{attribute 'qualified_only'}
VAR_GLOBAL CONSTANT
	DEFAULT_OPERATIONS_PER_CYCLE :UDINT := 2048;
END_VAR

(* stored: Version 1.1.0.1, ProductVersion 3.1.4026.8
   GVL GeneralParameters: Id {a36d7684-dab4-4a13-b2e9-9c2659f56638}, ParameterList True *)
